(* IEC 61131-3 sources: AxTestProject/LStandardLibrary/Signal Handling, 10 files *)

(* ---- BinSignal.st ---- *)
NAMESPACE stdLib.SignalHandling
    CLASS BinSignal

        VAR PRIVATE
            m_status : BinSignalStatus;
            m_Old : BOOL;
        END_VAR

        METHOD PUBLIC set : BinSignalStatus
            VAR_INPUT
                signal : BOOL;
                valid : BOOL := TRUE;
                default : BOOL := FALSE;
            END_VAR
            VAR_TEMP
                sig : BOOL;
            END_VAR
            IF (valid) THEN
                sig := signal;
                m_status.QBAD := FALSE;
            ELSE
                sig := default;
                m_status.QBAD := TRUE;
            END_IF;

            m_Status.QRis := sig AND NOT(m_Old);
            m_Status.QFal := NOT(sig) AND m_Old;

            m_Old := sig;
            m_status.Q := sig;

            set := m_status;
        END_METHOD

        METHOD PUBLIC Q : BOOL
            Q := m_status.Q;
        END_METHOD

        METHOD PUBLIC QRis : BOOL
            QRis := m_status.QRis;
        END_METHOD

        METHOD PUBLIC QFal : BOOL
            QFal := m_status.QFal;
        END_METHOD

        METHOD PUBLIC QBad : BOOL
            QBad := m_status.QBad;
        END_METHOD

        METHOD GetStatus : BinSignalStatus
            GetStatus := m_status;
        END_METHOD

    END_CLASS

    TYPE BinSignalStatus : STRUCT
            Q : BOOL;
            QRis : BOOL;
            QFal : BOOL;
            QBad : BOOL;
        END_STRUCT;
    END_TYPE

END_NAMESPACE

(* ---- Encoder.st ---- *)
NAMESPACE stdLib.SignalHandling
    CLASS Encoder
        VAR PRIVATE
            m_aOld : BOOL;
            m_bOld : BOOL;
            m_status : EncoderStatus;
        END_VAR

        // Reset encoder position to zero
        METHOD PUBLIC Reset
            m_status.position := DINT#0;
        END_METHOD

        //Set encoder to specific position
        METHOD PUBLIC Set
            VAR_INPUT
                position : DINT;
            END_VAR
                m_Status.position := position;
                ;
        END_METHOD

        //Evaluate encoder signals A and B
        METHOD PUBLIC evaluate
            VAR_INPUT
                a : BOOL;
                b : BOOL;
                aOOP : BinSignal;
                bOOP : BinSignal;
            END_VAR
            VAR_TEMP
                aRis : BOOL;
                bRis : BOOL;
                aFal : BOOL;
                bFal : BOOL;
            END_VAR

            IF (
                aOOP.QRis() AND NOT(bOOP.Q)
                OR
                aOOP.Q() AND bOOP.QRis()
                OR aOOP.QFal() AND bOOP.Q()

                OR NOT(a) AND bFal) THEN
                m_status.isInMotion := true;
                m_status.direction := false;
                m_status.position := m_status.position + DINT#1;
                m_status.increments := m_status.increments + DINT#1;

            aRis := a AND NOT(m_aOld);
            aFal := NOT(a) AND m_aOld;
            m_aOld := a;

            bRis := b AND NOT(m_bOld);
            bFal := NOT(b) AND m_bOld;
            m_bOld := b;

            //Forward detection
            IF (
                aRis AND NOT(b)
                OR a AND bRis
                OR aFal AND b
                OR NOT(a) AND bFal) THEN
                m_status.isInMotion := true;
                m_status.direction := false;
                m_status.position := m_status.position + DINT#1;
                m_status.increments := m_status.increments + DINT#1;
            //Reverse detection
            ELSIF
            (
                aRis AND b
                OR NOT(a) AND bRis
                OR aFal AND NOT(b)
                OR a AND bFal) THEN
                m_status.isInMotion := true;
                m_status.direction := true;
                m_status.position := m_status.position - DINT#1;
                m_status.increments := m_status.increments - DINT#1;
            ELSE
                m_status.isInMotion := false;
                m_status.direction := false;
            END_IF;

        END_METHOD

        METHOD PUBLIC GetStatus : EncoderStatus
            ;
            GetStatus := m_status;
            m_status.increments := DINT#0;
        END_METHOD

        METHOD PUBLIC SetInternals
            VAR_INPUT
                aOld : BOOL;
                bOld : BOOL;
            END_VAR
            m_aOld := aOld;
            m_bOld := bOld;
        END_METHOD

    END_CLASS

    TYPE EncoderStatus :
        STRUCT
            position : DINT;  // increments since last reset
            increments : DINT; // increments since last GetStatus-Call
            direction : BOOL; // 0: forward; 1: reverse
            isInMotion : BOOL; // encoder is in motion
        END_STRUCT;
    END_TYPE
END_NAMESPACE

(* ---- OnDelay.st ---- *)
NAMESPACE stdLib.Timer
    //##################################################################
    // Class: OnDelay
    //
    // Description: provides a on delay in OOP
    //##################################################################
    CLASS OnDelay
        VAR
            m_timeElapsed : DINT;
            m_status : Timerstatus;
            m_old : BOOL;
            m_isRunning : BOOL;
            m_PT : DINT;
            m_timeOld : DINT;
        END_VAR

        VAR PUBLIC
        END_VAR

        //##################################################################
        // Method Reset
        //
        // Reset a timer. Q will be reset to FALSE
        //##################################################################
        METHOD PUBLIC Reset
            m_isRunning := FALSE;
            m_status.Q := FALSE;
            m_status.ET := DINT#0;
            m_PT := DINT#0;
        END_METHOD

        METHOD PUBLIC Start
            VAR_INPUT
                PT : DINT;
                Retrigger : BOOL := false;
            END_VAR

            IF (retrigger OR NOT(m_isRunning)) THEN
                m_PT := PT;
                m_status.ET := m_PT;
                m_status.Q := FALSE;
                m_isRunning := TRUE;
            END_IF;
        END_METHOD

        METHOD PUBLIC Execute : BOOL

            VAR_EXTERNAL
            END_VAR

            VAR_INPUT
                sysLibTimer : DINT;
            END_VAR
            VAR_TEMP
                tTimeDifference : DINT;
            END_VAR

            tTimeDifference := ((sysLibTimer - m_timeOld) +  System.Const.MaxTimer()) MOD  System.Const.MaxTimer();
            m_timeOld := sysLibTimer;

            if (m_isRunning) then
                m_status.ET := m_status.ET - tTimeDifference;
            end_if;

            if (m_status.ET <= DINT#0 AND m_isRunning) then
                m_status.Q := true;
                m_isRunning := false;
            END_IF;
            Execute := m_status.Q;
        END_METHOD

        METHOD PUBLIC Q : BOOL
            Q := m_status.Q;
        END_METHOD

        METHOD PUBLIC GetStatus : Timerstatus
            VAR_INPUT
            END_VAR
            VAR_TEMP
            END_VAR
                GetStatus := m_status;
                ;
        END_METHOD

    END_CLASS

    TYPE Timerstatus :
        STRUCT
            Q : BOOL;
            ET : DINT;
        END_STRUCT;
    END_TYPE

END_NAMESPACE

(* ---- AnalogSignalTest.st ---- *)
NAMESPACE StdLibTesting.AnalogSignal

    {Test}
    FUNCTION EnableDisableLimiter
        VAR_INPUT
        END_VAR
        VAR_TEMP
            o : stdLib.SignalHandling.AnalogSignal;
            status : stdLib.SignalHandling.AnalogSignalStatus;
        END_VAR

        // Enable Limiter
        status := o.execute(signal := 100.0, enable := true);
        Assert_Equal_BOOL(expected := false, actual := status.LimiterIsEnabled);
        o.EnableLimiter(-200.0, 200.0);
        status := o.execute(signal := 100.0, enable := true);
        Assert_Equal_BOOL(expected := true, actual := status.LimiterIsEnabled);

        //disable limiter
        o.DisableLimiter();
        status := o.execute(signal := 100.0, enable := true);
        Assert_Equal_BOOL(expected := false, actual := status.LimiterIsEnabled);

    END_FUNCTION

// In Range
 {Test(av := 199, ll := -200, hl := 200, expQ := 199, expMax := 0, expMin := 0)}
 {Test(av := -199, ll := -200, hl := 200, expQ := -199, expMax := 0, expMin := 0)}
// Max Limit
 {Test(av := 200, ll := -200, hl := 200, expQ := 200, expMax := 1, expMin := 0)}
 {Test(av := 201, ll := -200, hl := 200, expQ := 200, expMax := 1, expMin := 0)}
// Min Limit
 {Test(av := -200, ll := -200, hl := 200, expQ := -200, expMax := 0, expMin := 1)}
 {Test(av := -201, ll := -200, hl := 200, expQ := -200, expMax := 0, expMin := 1)}

    FUNCTION CheckLimiter
        VAR_INPUT
            av : INT; //actual value
            ll : INT; //Lower Limit
            hl : INT; // higher limit
            expQ : INT; //expected Q
            expMax : INT; //expected MaxLimitReached
            expMin : INT; //expected MinLimitReached

        END_VAR
        VAR_TEMP
            o : stdLib.SignalHandling.AnalogSignal;
            status : stdLib.SignalHandling.AnalogSignalStatus;
            tAv : LREAL;
            tLL : LREAL;
            tHL : LREAL;
            tExpQ : LREAL;
            tMax : BOOL;
            tMin : BOOL;
        END_VAR

        tAv := INT_TO_LREAL(av);
        tLL := INT_TO_LREAL(ll);
        tHL := INT_TO_LREAL(hl);
        tExpQ := INT_TO_LREAL(expQ);
        tMax := expMax <> 0;
        tMin := expMin <> 0;

        // Enable Limiter
        o.EnableLimiter(tLL, tHL);

        // Max Limit reached
        status := o.execute(signal := tAv, enable := true);
        Assert_Equal_BOOL(expected := tMax, actual := status.MaxLimitReached);
        Assert_Equal_BOOL(expected := tMin, actual := status.MinLimitReached);
        Assert_Equal_LREAL(expected := tExpQ, actual := status.Q);
    END_FUNCTION

END_NAMESPACE

(* ---- BinOutputTest.st ---- *)
NAMESPACE StdLibTesting.BinOutput

    //-----------------------------------------------------------
    // test SetQ(value)
    //-----------------------------------------------------------
    {Test(value := 0, expect := 0)}
    {Test(value := 1, expect := 1)}
    FUNCTION TestSetQ
        VAR_INPUT
            value : INT;
            expect : INT;
        END_VAR

        VAR_TEMP
            o : stdLib.SignalHandling.BinOutput;
            tValue : BOOL;
            tExp : BOOL;
            tActual : BOOL;
        END_VAR

        tValue := value <> 0;
        tExp := expect <> 0;

        o.SetQ(value := tValue);
        Assert_Equal_BOOL(expected := tExp, actual := o.IsOn());
    END_FUNCTION

    //-----------------------------------------------------------
    // test SetOn
    //-----------------------------------------------------------
    {Test}
    FUNCTION SetOn
        VAR_TEMP
            o : stdLib.SignalHandling.BinOutput;
        END_VAR

        Assert_Equal_BOOL(expected := false, actual := o.IsOn());
        o.SetOn();
        Assert_Equal_BOOL(expected := true, actual := o.IsOn());
    END_FUNCTION

    //-----------------------------------------------------------
    // test SetOff
    //-----------------------------------------------------------
    {Test}
    FUNCTION SetOff

        VAR_TEMP
            o : stdLib.SignalHandling.BinOutput;
        END_VAR

        o.SetOn();
        Assert_Equal_BOOL(expected := true, actual := o.IsOn());
        o.SetOff();
        Assert_Equal_BOOL(expected := false, actual := o.IsOn());
    END_FUNCTION

    //-----------------------------------------------------------
    // test SetOff
    //-----------------------------------------------------------
    {Test}
    FUNCTION Toggle

        VAR_TEMP
            o : stdLib.SignalHandling.BinOutput;
        END_VAR

        Assert_Equal_BOOL(expected := false, actual := o.IsOn());
        o.Toggle();
        Assert_Equal_BOOL(expected := true, actual := o.IsOn());
        o.Toggle();
        Assert_Equal_BOOL(expected := false, actual := o.IsOn());
    END_FUNCTION

END_NAMESPACE

(* ---- BinSignalTest.st ---- *)
NAMESPACE StdLibTesting.BinSignal

    {Test(iSignal := 0, iEnable := 0, iDefault := 0, iExpQ := 0, iExpQBad := 1)}
    {Test(iSignal := 0, iEnable := 0, iDefault := 1, iExpQ := 1, iExpQBad := 1)}
    {Test(iSignal := 0, iEnable := 1, iDefault := 0, iExpQ := 0, iExpQBad := 0)}
    {Test(iSignal := 0, iEnable := 1, iDefault := 1, iExpQ := 0, iExpQBad := 0)}

    {Test(iSignal := 1, iEnable := 0, iDefault := 0, iExpQ := 0, iExpQBad := 1)}
    {Test(iSignal := 1, iEnable := 0, iDefault := 1, iExpQ := 1, iExpQBad := 1)}
    {Test(iSignal := 1, iEnable := 1, iDefault := 0, iExpQ := 1, iExpQBad := 0)}
    {Test(iSignal := 1, iEnable := 1, iDefault := 1, iExpQ := 1, iExpQBad := 0)}

    FUNCTION execute
        VAR_INPUT
            iSignal : INT;
            iEnable : INT;
            iDefault : INT;
            iExpQ : INT;
            iExpQBad : INT;
        END_VAR

        VAR_TEMP
            o : stdLib.SignalHandling.BinSignal;
            status : stdLib.SignalHandling.BinSignalStatus;
            tSignal : BOOL;
            tEnable : BOOL;
            tDefault : BOOL;
            tExpQ : BOOL;
            tExpQBad : BOOL;
        END_VAR

        tSignal := iSignal <> 0;
        tEnable := iEnable <> 0;
        tDefault := iDefault <> 0;
        tExpQ := iExpQ <> 0;
        tExpQBad := iExpQBad <> 0;

        status := o.set(signal := tSignal, valid := tEnable, default := tDefault);
        Assert_Equal_BOOL(expected := tExpQ, actual := status.Q);
        ;
            ;
    END_FUNCTION

    {Test(iSignal := 1, iEnable := 1, iDefault := 0, iExpQ := 1, iExpQRis := 1, iExpQFal := 0, iTestFallingEdge := 0)}
    {Test(iSignal := 0, iEnable := 1, iDefault := 0, iExpQ := 0, iExpQRis := 0, iExpQFal := 1, iTestFallingEdge := 1)}

    FUNCTION QRis
        VAR_INPUT
            iSignal : INT;
            iEnable : INT;
            iDefault : INT;
            iExpQ : INT;
            iExpQRis : INT;
            iExpQFal : INT;
            iTestFallingEdge : INT;
        END_VAR
        VAR_TEMP
            o : stdLib.SignalHandling.BinSignal;
            status : stdLib.SignalHandling.BinSignalStatus;
            tSignal : BOOL;
            tEnable : BOOL;
            tDefault : BOOL;
            tExpQ : BOOL;
            tExpQRis : BOOL;
            tExpQFal : BOOL;
            tTestFallingEdge : BOOL;
        END_VAR

        tSignal := iSignal <> 0;
        tEnable := iEnable <> 0;
        tDefault := iDefault <> 0;
        tExpQ := iExpQ <> 0;
        tExpQRis := iExpQRis <> 0;
        tExpQFal := iExpQFal <> 0;
        tTestFallingEdge := iTestFallingEdge <> 0;

        if (tTestFallingEdge) then
            status := o.set(signal := true, valid := tEnable, default := tDefault);
        END_IF;

        status := o.set(signal := tSignal, valid := tEnable, default := tDefault);
        Assert_Equal_BOOL(expected := tExpQ, actual := status.Q);
        Assert_Equal_BOOL(expected := tExpQRis, actual := status.QRis);
        Assert_Equal_BOOL(expected := tExpQFal, actual := status.QFal);

        status := o.set(signal := tSignal, valid := tEnable, default := tDefault);
        Assert_Equal_BOOL(expected := tExpQ, actual := status.Q);
        Assert_Equal_BOOL(expected := false, actual := status.QRis);
        Assert_Equal_BOOL(expected := false, actual := status.QFal);
    END_FUNCTION
END_NAMESPACE

(* ---- EncoderTest.st ---- *)
NAMESPACE StdLibTesting.Encoder

    {Test}
    FUNCTION Reset
        VAR_INPUT
        END_VAR
        VAR_TEMP
            o : stdLib.SignalHandling.Encoder;
            status : stdLib.SignalHandling.EncoderStatus;
        END_VAR

        o.Set(DINT#555);
        status := o.GetStatus();
        Assert_Equal_DINT(expected := DINT#555, actual := status.position);
        o.Reset();
        status := o.GetStatus();
        Assert_Equal_DINT(expected := DINT#0, actual := status.position);
        Assert_Equal_DINT(expected := DINT#0, actual := status.increments);
        ;
            ;
    END_FUNCTION

    {Test( aOld := 0, a := 0, bOld := 0, b := 0, dir := 0, pos := 0)}
    {Test( aOld := 1, a := 1, bOld := 1, b := 1, dir := 0, pos := 0)}

    {Test( aOld := 0, a := 1, bOld := 0, b := 0, dir := 0, pos := 1)}
    {Test( aOld := 1, a := 0, bOld := 1, b := 1, dir := 0, pos := 1)}
    {Test( aOld := 1, a := 1, bOld := 0, b := 1, dir := 0, pos := 1)}
    {Test( aOld := 0, a := 0, bOld := 1, b := 0, dir := 0, pos := 1)}

    {Test(a := 1, b := 1, aOld := 0, bOld := 1, dir := 1, pos := -1)}
    {Test(a := 0, b := 1, aOld := 0, bOld := 0, dir := 1, pos := -1)}
    {Test(a := 0, b := 0, aOld := 1, bOld := 0, dir := 1, pos := -1)}
    {Test(a := 1, b := 0, aOld := 1, bOld := 1, dir := 1, pos := -1)}

    FUNCTION EncoderDirection
        VAR_INPUT
            a : INT;
            b : INT;
            aOld : INT;
            bOld : INT;
            dir : INT;
            pos : INT;
        END_VAR
        VAR
            tA : BOOL;
            tB : BOOL;
            tAOld : BOOL;
            tBOld : BOOL;
            tDir : BOOL;
            o : stdLib.SignalHandling.Encoder;
            status : stdLib.SignalHandling.EncoderStatus;
        END_VAR
        tA := a <> 0;
        tB := b <> 0;
        tAOld := aOld <> 0;
        tBold := bOld <> 0;
        tDir := dir <> 0;
        o.SetInternals(aOld := tAOld, bOld:= tBold);
        o.Evaluate(tA, tB);
        status := o.GetStatus();

        Assert_Equal_BOOL(expected := tDir, actual := status.direction);
        Assert_Equal_DINT(expected := INT_TO_DINT(pos), actual := status.position);
        Assert_Equal_DINT(expected := INT_TO_DINT(pos), actual := status.increments);

        status := o.GetStatus();
        Assert_Equal_DINT(expected := INT_TO_DINT(pos), actual := status.position);
        Assert_Equal_DINT(expected := DINT#0, actual := status.increments);
        ;
    END_FUNCTION

//################################################################################
//
//################################################################################
    {Test( a_t0 := 0, b_t0 := 0, a_t1 := 0, b_t1 := 0, dir := 0, pos := 0)}
    {Test( a_t0 := 0, b_t0 := 0, a_t1 := 1, b_t1 := 0, dir := 0, pos := 1)}
    {Test( a_t0 := 1, b_t0 := 0, a_t1 := 1, b_t1 := 0, dir := 0, pos := 0)}
    {Test( a_t0 := 1, b_t0 := 0, a_t1 := 1, b_t1 := 1, dir := 0, pos := 1)}
    {Test( a_t0 := 1, b_t0 := 1, a_t1 := 1, b_t1 := 1, dir := 0, pos := 0)}
    {Test( a_t0 := 1, b_t0 := 1, a_t1 := 0, b_t1 := 1, dir := 0, pos := 1)}
    {Test( a_t0 := 0, b_t0 := 1, a_t1 := 0, b_t1 := 1, dir := 0, pos := 0)}
    {Test( a_t0 := 0, b_t0 := 1, a_t1 := 0, b_t1 := 0, dir := 0, pos := 1)}

    {Test( a_t0 := 0, b_t0 := 0, a_t1 := 0, b_t1 := 1, dir := 1, pos := -1)}
    {Test( a_t0 := 0, b_t0 := 1, a_t1 := 1, b_t1 := 1, dir := 1, pos := -1)}
    {Test( a_t0 := 1, b_t0 := 1, a_t1 := 1, b_t1 := 0, dir := 1, pos := -1)}
    {Test( a_t0 := 1, b_t0 := 0, a_t1 := 0, b_t1 := 0, dir := 1, pos := -1)}

    FUNCTION EncoderDirection_new
        VAR_INPUT
            a_t1 : INT;
            b_t1 : INT;
            a_t0 : INT;
            b_t0 : INT;
            dir : INT;
            pos : INT;
        END_VAR
        VAR
            tA_t1 : BOOL;
            tB_t1 : BOOL;
            tA_t0 : BOOL;
            tB_t0 : BOOL;
            tDir : BOOL;
            o : stdLib.SignalHandling.Encoder;
            status : stdLib.SignalHandling.EncoderStatus;
        END_VAR
        tA_t1 := a_t1 <> 0;
        tB_t1 := b_t1 <> 0;
        tA_t0 := a_t0 <> 0;
        tB_t0 := b_t0 <> 0;
        tDir := dir <> 0;
        o.Evaluate(tA_t0, tB_t0);
        o.Evaluate(tA_t1, tB_t1);
        status := o.GetStatus();

        Assert_Equal_BOOL(expected := tDir, actual := status.direction);
        Assert_Equal_DINT(expected := INT_TO_DINT(pos), actual := status.position);
        Assert_Equal_DINT(expected := INT_TO_DINT(pos), actual := status.increments);

        status := o.GetStatus();
        Assert_Equal_DINT(expected := INT_TO_DINT(pos), actual := status.position);
        Assert_Equal_DINT(expected := DINT#0, actual := status.increments);
        ;
    END_FUNCTION
END_NAMESPACE

(* ---- OnDelayTest.st ---- *)
NAMESPACE StdLibTesting.Encoder

    {Test}
    FUNCTION Start_Q
        VAR_INPUT
        END_VAR
        VAR_TEMP
            o : stdLib.Timer.OnDelay;
            status : stdLib.Timer.TimerStatus;
        END_VAR

        o.Start(PT := DINT#5000);
        Assert_Equal_BOOL(expected := false, actual := o.Q());
        Assert_Equal_DINT(expected := DINT#5000, actual := o.GetStatus().ET);
    END_FUNCTION

    {Test}
    FUNCTION Start_Q_retrigger
        VAR_INPUT
        END_VAR
        VAR_TEMP
            o : stdLib.Timer.OnDelay;
            status : stdLib.Timer.TimerStatus;
        END_VAR

        o.Start(PT := DINT#5000, retrigger := true);
        Assert_Equal_BOOL(expected := false, actual := o.Q());
        Assert_Equal_DINT(expected := DINT#5000, actual := o.GetStatus().ET);
    END_FUNCTION

        {Test}
    FUNCTION Start_Q_TwoStarts
        VAR_INPUT
        END_VAR
        VAR_TEMP
            o : stdLib.Timer.OnDelay;
            status : stdLib.Timer.TimerStatus;
        END_VAR

        o.Start(PT := DINT#5000);
        Assert_Equal_BOOL(expected := false, actual := o.Q());
        Assert_Equal_DINT(expected := DINT#5000, actual := o.GetStatus().ET);
        o.Start(PT := DINT#9000);
        Assert_Equal_BOOL(expected := false, actual := o.Q());
        Assert_Equal_DINT(expected := DINT#5000, actual := o.GetStatus().ET);
    END_FUNCTION

    {Test}
    FUNCTION Start_Q_TwoStartsRetrig
        VAR_INPUT
        END_VAR
        VAR_TEMP
            o : stdLib.Timer.OnDelay;
            status : stdLib.Timer.TimerStatus;
        END_VAR

        o.Start(PT := DINT#5000);
        Assert_Equal_BOOL(expected := false, actual := o.Q());
        Assert_Equal_DINT(expected := DINT#5000, actual := o.GetStatus().ET);
        o.Start(PT := DINT#9000, retrigger := true);
        Assert_Equal_BOOL(expected := false, actual := o.Q());
        Assert_Equal_DINT(expected := DINT#9000, actual := o.GetStatus().ET);
    END_FUNCTION
END_NAMESPACE

(* ---- BinOutput.st ---- *)
NAMESPACE stdLib.SignalHandling
    CLASS BinOutput

        VAR
            m_State : BOOL;
        END_VAR

        METHOD PUBLIC RefToOutput
            VAR_OUTPUT
                Q : BOOL;
            END_VAR
            Q:= m_state;
        END_METHOD

        METHOD PUBLIC SetQ
            VAR_INPUT
                value : BOOL;
            END_VAR
            m_State := value;
        END_METHOD

        METHOD PUBLIC SetOn
            m_State := TRUE;
        END_METHOD

        METHOD PUBLIC SetOff
            m_State := FALSE;
        END_METHOD

        METHOD PUBLIC Toggle
            m_state := NOT(m_state);
        END_METHOD

        METHOD PUBLIC IsOn : BOOL
            IsOn := m_state;
        END_METHOD

    END_CLASS
END_NAMESPACE

(* ---- ClockGenerator.st ---- *)
NAMESPACE stdLib.Timer
    CLASS ClockGenerator

    VAR PRIVATE
        m_timer1 : stdLib.Timer.OnDelay;
        m_timer2 : stdLib.Timer.OnDelay;
        m_isRunning : BOOL;
        m_q : BOOL;
    END_VAR

    METHOD PUBLIC Execute
        VAR_INPUT
            pulse : DINT;
            pause : DINT;
            sysLibTimer : DINT;
        END_VAR

            m_timer1.Execute(sysLibTimer);
            m_timer2.Execute(sysLibTimer);

            IF (m_timer2.Q() OR not(m_isRunning)) THEN
                m_timer1.Start(PT := pulse);
                m_timer2.Reset();
                m_isRunning := true;
                m_q := true;
            END_IF;

            if (m_timer1.Q() ) then
                m_timer2.Start(PT:=pause);
                m_timer1.Reset();
                m_q := false;
            End_if;
    END_METHOD

    METHOD PUBLIC Q : BOOL
        Q := m_q;
    END_METHOD

    END_CLASS

END_NAMESPACE
